{attribute 'qualified_only'}
VAR_GLOBAL
	AllShortContactEngaged	: BOOL;
	AllDumpRelaysOpen		: BOOL;
	AllChargeRelaysClosed	: BOOL;
	
END_VAR

(* stored: Version 1.1.0.1, ProductVersion 3.1.4024.11
   GVL Permissives_DB: Id {c05a4b99-99cd-4605-96e2-a97127a00965} *)
